Staubli VAL3: default.pjx

--- default.pjx ---
Parameters version=s7.9.1 stackSize=5000 millimeterUnit=true
Program file=start.pgx
Program file=stop.pgx
Data file=default.dtx

--- start.pgx ---
program start()
begin
end
